PROGRAM P_Demo_NT_GetTime
VAR
    fbNT_GetTime : NT_GetTime; // NT_GetTime 实例
    bRead        : BOOL := FALSE;
    stTimeOut    : TIMESTRUCT;
    bBusy_       : BOOL;
    bErrFlag     : BOOL;
    nErrCode     : UDINT;
END_VAR

// =============================================================================
// 场景：一次性读 Windows 时间。
// 价值：标准 ADS 调用。
// 验证：改 bRead := TRUE，观察 stTimeOut 装载时间且与桌面时钟一致。
// 验证步骤：
//   1. 右键 PLC 项目下 POUs 文件夹 → Add → Existing Item → 选本 .TcPOU 文件
//   2. 引用 Tc2_Utilities（References → Add library）
//   3. 编译 → 登录 → 运行；按上方『验证』行的指示在线写值观察
// =============================================================================

fbNT_GetTime(
    NETID := '', START := bRead, TMOUT := DEFAULT_ADS_TIMEOUT,
    TIMESTR => stTimeOut, BUSY => bBusy_, ERR => bErrFlag, ERRID => nErrCode
);

END_PROGRAM

(* stored: Version 1.1.0.1, ProductVersion 3.1.4024.5
   POU P_Demo_NT_GetTime: Id {2bf6d160-eef7-5691-924d-277595f1ba7e}, SpecialFunc None *)
